(* PLC project Function Block Example.project, CODESYS CODESYS V3.5 SP20 Patch 1 *)
(* stored: creationDateTime 2025-05-22T17:28:10.8991994, modificationDateTime 2025-05-22T17:27:01.9379103 *)

PROGRAM Main
  VAR
    MyMotorInstance1 : Motor;
    MyMotorInstance2 : Motor;
    MyMotorInstance3 : Motor;
  END_VAR

                    
MyMotorInstance1();
MyMotorInstance2();
MyMotorInstance3();
                  
END_PROGRAM

FUNCTION_BLOCK Motor

                    
// Motor control logic here
                  
END_FUNCTION_BLOCK

CONFIGURATION Device
  RESOURCE Application ON PLC
    TASK MainTask(INTERVAL := T#20ms, PRIORITY := 1);
    PROGRAM Main WITH MainTask : Main;
  END_RESOURCE
END_CONFIGURATION
